// TIA Portal V19 export
TYPE "LEXCHANGETRAY_typePlasticEm5_toRollerReq"
// stored: Access Published
   STRUCT
      inFeedReq : Bool;
      outFeedReq : Bool;   // 请求排料
   END_STRUCT;
END_TYPE
